(****************************************************************
NAME:			FB_DecoupleAxis
DATA:			2017.2.24
VERSION:		1.0.0
DESCRIPTION:	FB_DecoupleAxis
HISTORY:
				2017.2.16		NEW

***************************************************************)
FUNCTION_BLOCK FB_DecoupleAxis
VAR_INPUT
	Execute:BOOL;
	Reset:BOOL;
END_VAR
VAR_OUTPUT
	FbID:DINT:=1001;
	State:DINT;
	Busy:BOOL;
	OutGear:BOOL;
	Error:BOOL;
	ErrorID:DINT;
END_VAR
VAR
	Top_MC_GearOut: MC_GearOut;
	Bottom_MC_GearOut: MC_GearOut;
	fb_ton: TON;
END_VAR

IF Execute THEN
Busy:=TRUE;
fb_ton(PT:=t#0.1s);
CASE State OF
	0:	(*Decouple Check*)
		IF  LeftTopLin.NcToPlc.CoupleState=0 AND RightTopLin.NcToPlc.CoupleState=0
			AND LeftBottomLin.NcToPlc.CoupleState=0 AND RightBottomLin.NcToPlc.CoupleState=0 THEN	
			State:=88;
		ELSIF LeftTopLin.NcToPlc.CoupleState<>1 AND RightTopLin.NcToPlc.CoupleState<>3
			AND LeftBottomLin.NcToPlc.CoupleState<>1 AND RightBottomLin.NcToPlc.CoupleState<>3 THEN		
			ErrorID:=1;
			State:=-100;
		ELSIF Top_MC_GearOut.Error OR Bottom_MC_GearOut.Error THEN		(*FB ´íÎó*)
			ErrorID:=2;
			State:=99;
		ELSIF LeftTopLin.NcToPlc.CoupleState=1 AND RightTopLin.NcToPlc.CoupleState=3
			AND LeftBottomLin.NcToPlc.CoupleState=1 AND RightBottomLin.NcToPlc.CoupleState=3 THEN		
			State:=1;
		END_IF
	1:	(*Decouple*)
		IF LeftTopLin.NcToPlc.CoupleState=1 AND RightTopLin.NcToPlc.CoupleState=3
			AND LeftBottomLin.NcToPlc.CoupleState=1 AND RightBottomLin.NcToPlc.CoupleState=3 THEN		
			Top_MC_GearOut.Execute:=TRUE;
			Bottom_MC_GearOut.Execute:=TRUE;
			A_DecoupleMC();
			fb_ton.IN:=TRUE;
		ELSIF LeftTopLin.NcToPlc.CoupleState=0 AND RightTopLin.NcToPlc.CoupleState=0
			AND LeftBottomLin.NcToPlc.CoupleState=0 AND RightBottomLin.NcToPlc.CoupleState=0 THEN	
			State:=88;
		ELSE
			ErrorID:=3;
			State:=-100;
		END_IF
	2:	(*Decouple Wait*)
		A_DecoupleMC();
		IF NOT Top_MC_GearOut.Done OR NOT Bottom_MC_GearOut.Done THEN	
			IF NOT fb_ton.Q THEN
				State:=2;
			ELSE
				ErrorID:=4;
				State:=99;
			END_IF
		ELSIF Top_MC_GearOut.Done AND Bottom_MC_GearOut.Done
			AND LeftTopLin.NcToPlc.CoupleState=0 AND RightTopLin.NcToPlc.CoupleState=0
			AND LeftBottomLin.NcToPlc.CoupleState=0 AND RightBottomLin.NcToPlc.CoupleState=0 THEN		
			State:=88;
		ELSE
			ErrorID:=5;
			State:=-100;
		END_IF
	88:	(*Done*)
		Execute:=FALSE;
		State:=0;
		Busy:=FALSE;
		OutGear:=TRUE;
		Error:=FALSE;
		ErrorID:=0;
		Top_MC_GearOut.Execute:=FALSE;
		Bottom_MC_GearOut.Execute:=FALSE;
		A_DecoupleMC();
		fb_ton.IN:=FALSE;
	99:	(*FB Error*)
		Execute:=FALSE;
		State:=99;
		Busy:=FALSE;
		OutGear:=FALSE;
		Error:=TRUE;
		Top_MC_GearOut.Execute:=FALSE;
		Bottom_MC_GearOut.Execute:=FALSE;
		A_DecoupleMC();
		fb_ton.IN:=FALSE;
	-100:	(*EStop Error*)
		FB_PlcEmergencyStop();
		Execute:=FALSE;
		State:=-100;
		Busy:=FALSE;
		OutGear:=FALSE;
		Error:=TRUE;
		Top_MC_GearOut.Execute:=FALSE;
		Bottom_MC_GearOut.Execute:=FALSE;
		A_DecoupleMC();
		fb_ton.IN:=FALSE;

END_CASE
END_IF
IF Reset THEN
		Execute:=FALSE;
		State:=0;
		Busy:=FALSE;
		OutGear:=FALSE;
		Error:=FALSE;
		ErrorID:=0;
		Top_MC_GearOut.Execute:=FALSE;
		Bottom_MC_GearOut.Execute:=FALSE;
		A_DecoupleMC();
		fb_ton.IN:=FALSE;
		Reset:=FALSE;
END_IF

ACTION A_DecoupleMC:
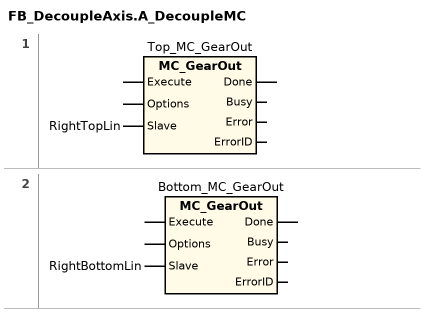
// NETWORK 1
Top_MC_GearOut(Slave := RightTopLin); // MC_GearOut

// NETWORK 2
Bottom_MC_GearOut(Slave := RightBottomLin); // MC_GearOut
END_ACTION

END_FUNCTION_BLOCK

(* stored: Version 1.1.0.1, ProductVersion 3.1.4024.6
   POU FB_DecoupleAxis: Id {2e8fd5f4-f61e-4c5b-a0b0-e83b4112a9ea}, SpecialFunc None
   Action A_DecoupleMC: Id {464c74fe-3945-4d3f-abbc-f0c57fbc5f90} *)
